FUNCTION_BLOCK FB 52
TITLE = Motor with 6 digital input
//  
//COPYRIGHT:    (C) 1997  BUHLER AG, CH-9240 UZWIL,  SWITZERLAND
//
//PRODUCT:      GCS7
//
//TITLE:        FB 50 MACHINE-CONTROL:Motor with 6 Digital input 
//              GCPROVB Revision >=12
// 
//-------------------------------------------------------------------------
//
//IDENT:        AUTHOR:             DEPT:                       DATE:
//FB50.8.6      A.Egli              BASE                        10-Apr-2008
//              - Init if download DB
//              - Condition MonX.InLocal 
//FB50.8.5      Ph. Engler          GP92                        23-Aug-2007
//              Machine status: StStarting how long the monitoring elements
//FB50.8.5      Ph. Engler          GP92                        23-Aug-2007
//              Machine status: StStarting how long the monitoring elements
//                              aren't in the correct status
//FB50.8.4      A.Egli              CT3                         20-Feb-2006
//              EBM-Test procedure: - Include als the EBMInput to the test
//                                  - Manual and local mode also integrated 
//              (Tested Ph.Engler, GP92,24-Aug-2005 )
//FB50.8.3      A.Egli              CT3                         09-Mar-2005
//              Send CmdFaultReset only with positve edge to elements  
//FB50.8.2      A.Egli              CT3                         20-Sep-2004 
//              Delay time before and between 2 single tests of EBM  
//FB50.8.1      A.Egli              CT3                         20-Jul-2004
//              tmpLenDyn is 12 and not 10
//FB50.8.0      A.Egli              CT3                         25-Mai-2004
//              ParMon4IsSM
//FB50.7.6      A.Egli              CT3                         15-Apr-2004
//              Test with Hardware 
//FB50.7.5      A.Egli              CT3                         18-Mar-2004
//              InpControlEBM 
//FB50.7.4      K. Tischer          CT3                         13-Feb-2004
//              interlocking without Mon1 
//FB50.7.3      K. Tischer          CT3                         30-Jan-2004
//              Correct monitoring Mon4 
//FB50.7.2      K. Tischer          CT3                         14-Jan-2004
//              Revision=11 
//FB50.7.1      K. Tischer          CT3                         02-Dec-2003
//              new 6 DI and supported EBM3003 
//FB50.7.0      K. Tischer          CT3                         01-Dec-2003
//              new 6 DI and supported EBM3003 
//FB50.6.2      A. Egli             CT3                         22-Sep-2003
//              Interlocking Mon4.StFalse when Mon4 is HL
//FB50.6.1      A. Egli             CT3                         16-Mai-2003
//              Interlocking if Mon1 is HL
//              Send CmdOff to Motor
//FB50.6.0      A. Egli             CT3                         17-Jun-2002
//              New Release with one block 
//              Interlocking if Mon1 is HL
//FB50.5.0      A. Egli             CT3                          1-Feb-2002
//              -HLInlet renamed as Mon4
//              -ParMon4StopByFault,ParMon4IsLS
//FB50.4.0      A. Egli             CT3                         15-Jan-2002
//              HLIntet as Warning Element
//FB50.3.1      A. Egli             CT3                         23-Oct-2001
//              Manual Mode: no interlocking with InSeqStop
//FB50.3.0      A. Egli             CT3                         11-Oct-1999
//              Local data reduced 
//FB50.2C       A. Egli             CT3                         03-Juni-1999
//              Manual Mode
//FB50.2B       K. Tischer          MU664                       06-Mrz-1999
//              CC FC2 not UC FC2
//FB50.2A       A. Egli             CT3                         04-Mai-1998
//              StFault = StCode 32
//FB50.1A       A.Egli              AEE61                       5-Jul-1997
//              1st Release in S7
//
//-------------------------------------------------------------------------
//
//PURPOSE:      MANUAL : see [LL.M4IxxMAN]
//
//RESTRICTIONS: S7
//
//              GCPROVB Revision >=5
//-------------------------------------------------------------------------
//
AUTHOR : EA
FAMILY : GCS7LL
NAME : M_6DI
VERSION : 8.6
VAR
  Ma : UDT 20500;
  Mon1 : FB 14;	//Element Mon 1 optional
  Mon2 : FB 14;	//Element Mon 2
  Mon3 : FB 14;	//Element Mon 3 optional
  Mon4 : FB 14;	//Element Mon 4 optional
  Mon5 : FB 14;	//Element Mon 5 optional [7.0]
  Mon6 : FB 14;	//Element Mon 6 optional [7.0]
  Motor : FB 12;	//Element Motor
END_VAR
VAR_TEMP
  tmpFaultStop : BOOL ;
  tmpFaultSum : BOOL ;
  tmpEnable : BOOL ;
  tmpLocal : BOOL ;
  tmpLenDyn : INT ;
  tmpOK : BOOL ;
  tmpTestTime : INT ;
  tmpMonElOk : BOOL ;
END_VAR
BEGIN
NETWORK
TITLE =
      L     12;
      T     #tmpLenDyn;	//[8.1]
NETWORK
TITLE = PC Control
//=== Test Object number =====================
      L     DB3.DBW 50;	//PCControl.ObjectNo
      L     DIW [AR2,P#8.0];	//Input ObjectNo
      <>I;
      JC    aEnd;
//=== Test OType      ========================
      L     2050;	//Input object type
      L     DB3.DBW 48;	//PCControl.ObjectType
      <>I;
      JC    aEnd;
//=== Test Handshake =========================
      A     DB3.DBX 43.3;	// Handshake.FExamine
      JC    aExa;
      A     DB3.DBX 43.0;	// Handshake.FDefineCmd
      O     DB3.DBX 43.1;	// Handshake.FDefinePara
      JC    aCmd;
aIni: L     2;	// FcInit
      UC    FC 3;
      JU    aEnd;
// Write new commands from PC to Interface of group 
aCmd: A     DB3.DBX 53.0;	//Cmd1[8]=CmdOff
      S     DIX [AR2,P#3.0];
      A     DB3.DBX 53.1;	//Cmd1[9]=CmdOn
      S     DIX [AR2,P#3.1];
      A     DB3.DBX 53.2;	//Cmd1[10]=CmdNext
      S     DIX [AR2,P#3.2];
      A     DB3.DBX 53.3;	//Cmd1[11]=CmdFaultReset
      S     DIX [AR2,P#3.3];
      A     DB3.DBX 53.5;	//Cmd1[13]=CmdManualOn
      S     DIX [AR2,P#3.5];
      A     DB3.DBX 52.6;	//Cmd1[6]=CmdManSlowOn
      S     DIX [AR2,P#221.6];
      A     DB3.DBX 52.7;	//Cmd1[7]=CmdManRevOn
      S     DIX [AR2,P#221.7];
      A     DB3.DBX 55.5;	//Cmd2[13]=CmdManualOff
      R     DIX [AR2,P#3.5];
      A     DB3.DBX 54.6;	//Cmd2[6]=CmdManSlowOff
      R     DIX [AR2,P#221.6];
      A     DB3.DBX 54.7;	//Cmd2[7]=CmdManRevOff
      R     DIX [AR2,P#221.7];
      JU    aIni;
aExa: TAR2;	// Address Dynamic datas
      T     DB3.DBD 24;	// -->PCControl.GC.InDynAddr
      L     #tmpLenDyn;	// Length Dynamic data
      T     DB3.DBW 22;	// -->PCControl.GC.InDynLen
      L     0;
      T     DB3.DBD 30;	// -->PCControl.GC.InParaAddr
      T     DB3.DBW 28;	// -->PCControl.GC.InParaLen
      L     1;	// Code FcExamine
      UC    FC 3;
      L     12;	//Revision
      T     DB3.DBW 34;
aEnd: NOP   0;
NETWORK
TITLE = function test [7.0]
      L     720;	//[8.2] 
      T     #tmpTestTime;	//[8.2] 
      AN    DIX [AR2,P#11.5];
      JC    FCT0;
      A     DIX [AR2,P#3.4];
      AN    DIX [AR2,P#3.5];
      =     #tmpLocal;
      L     0;
      L     DIW [AR2,P#6.0];
      >=I;
      O     DIX [AR2,P#3.6];
      R     DIX [AR2,P#4.1];
      R     DIX [AR2,P#4.2];
      R     DIX [AR2,P#4.3];
      R     DIX [AR2,P#3.6];
      L     #tmpTestTime;	//s = 12min 
      JC    FCT;
      AN    DIX [AR2,P#221.2];	//[8.2] 
      AN    DIX [AR2,P#221.5];	//[8.2] 
      AN    DIX [AR2,P#4.3];	//[8.2] 
      L     #tmpTestTime;	//[8.2] 
      JC    FCT;	//[8.2] 
      L     DIW [AR2,P#6.0];
      AN    M 10.5;	// Gr.OutTick1s
      JC    FCT;
      +     -1;
FCT:  T     DIW [AR2,P#6.0];
// function test SM
      L     #tmpTestTime;	//[8.2] 
      L     DIW [AR2,P#6.0];	//[8.2] 
      -I;	//[8.2] 
      L     35;	//[8.2] 
      >=I;	//[8.2] 
      A     DIX [AR2,P#2.6];	//[7.5]
      AN    DIX [AR2,P#4.7];	//[7.5]
      AN    DIX [AR2,P#5.4];	//[7.5]
      O     DIX [AR2,P#4.6];	//[7.5]
      AN    DIX [AR2,P#4.3];
      AN    DIX [AR2,P#15.4];
      AN    DIX [AR2,P#5.0];	//[8.2]
      =     DIX [AR2,P#4.6];
// function test ok SM
      A     DIX [AR2,P#4.6];
      A(;
      ON    DIX [AR2,P#184.6];
      ON    DIX [AR2,P#10.4];
      );
      AN    DIX [AR2,P#2.6];	//[7.5]
      =     #tmpOK;	//[7.5]
      A     #tmpOK;	//[7.5]
      AN    DIX [AR2,P#4.3];	//[7.5]
      S     DIX [AR2,P#4.3];
      S     DIX [AR2,P#2.5];	//[7.5]
      JCN   BTJ1;	//[8.2] 
      L     #tmpTestTime;	//[8.2] s = 12min 
      T     DIW [AR2,P#6.0];	//[8.2] 
BTJ1: NOP   0;	//[8.2] 
// function test BM top
      L     #tmpTestTime;	//[8.2] s = 12min 
      L     DIW [AR2,P#6.0];	//[8.2] 
      -I;	//[8.2] 
      L     5;	//[8.2] 
      >=I;	//[8.2] 
      AN    DIX [AR2,P#4.7];	//[7.5]
      A     DIX [AR2,P#2.6];	//[7.5]
      AN    DIX [AR2,P#5.4];	//[7.5]
      O     DIX [AR2,P#4.4];	//[7.5]
      AN    DIX [AR2,P#4.1];
      A     DIX [AR2,P#4.3];	//[7.6]
      AN    DIX [AR2,P#15.4];
      =     DIX [AR2,P#4.4];
// function test ok
      A     DIX [AR2,P#4.4];
      AN    DIX [AR2,P#48.6];
      AN    DIX [AR2,P#2.6];	//[7.5]
      =     #tmpOK;	//[7.5]
      A     #tmpOK;	//[7.5]
      AN    DIX [AR2,P#4.1];	//[7.5]
      S     DIX [AR2,P#4.1];
      S     DIX [AR2,P#2.5];	//[7.5]
      JCN   BTJ2;	//[8.2] 
      L     #tmpTestTime;	//[8.2] s = 12min 
      T     DIW [AR2,P#6.0];	//[8.2] 
BTJ2: NOP   0;	//[8.2] 
// function test BM Bottom
      L     #tmpTestTime;	//[8.2] s = 12min 
      L     DIW [AR2,P#6.0];	//[8.2] 
      -I;	//[8.2] 
      L     5;	//[8.2] 
      >=I;	//[8.2] 
      A     DIX [AR2,P#2.6];	//[7.5]
      AN    DIX [AR2,P#4.7];	//[7.5]
      AN    DIX [AR2,P#5.4];	//[7.5]
      O     DIX [AR2,P#4.5];	//[7.5]
      AN    DIX [AR2,P#4.2];
      A     DIX [AR2,P#4.1];
      A     DIX [AR2,P#4.3];	//[7.6]
      AN    DIX [AR2,P#15.4];
      =     DIX [AR2,P#4.5];
// function test ok BM Bottom 
      A     DIX [AR2,P#4.5];
      A(;
      ON    DIX [AR2,P#116.6];
      ON    DIX [AR2,P#10.2];
      );
      AN    DIX [AR2,P#2.6];	//[7.5]
      =     #tmpOK;	//[7.5]
      A     #tmpOK;	//[7.5]
      AN    DIX [AR2,P#4.2];	//[7.5]
      S     DIX [AR2,P#4.2];
      S     DIX [AR2,P#2.5];	//[7.5]
FCT0: NOP   0;
NETWORK
TITLE = Interlocking
//===Global Group Orders===
      A     M 12.5;	//Gr.OutManualOn
      S     DIX [AR2,P#3.5];
      A     M 12.4;	//Gr.OutManualOff
      R     DIX [AR2,P#3.5];
      A     DIX [AR2,P#3.5];
      S     M 13.5;	//Gr.InManual
// 
      A     M 12.3;	// OutFaultReset
      S     DIX [AR2,P#3.3];
//--- Fault----
      A     DIX [AR2,P#10.7];
      A     DIX [AR2,P#17.4];
      O     DIX [AR2,P#51.4];
      O     DIX [AR2,P#85.4];
      O(;	//[5.0]
      A     DIX [AR2,P#11.3];	//[5.0]
      O     DIX [AR2,P#11.6];	//[8.0]
      O     DIX [AR2,P#11.5];	//[7.6]
      A     DIX [AR2,P#119.4];	//[5.0]
      );	//[5.0]
      O     DIX [AR2,P#153.4];	//[7.0]
      O     DIX [AR2,P#187.4];	//[7.0]
      =     #tmpFaultStop;
      A     DIX [AR2,P#119.4];	//[4.0]
      AN    DIX [AR2,P#11.2];	//[4.0]
      O     DIX [AR2,P#17.4];
      O     DIX [AR2,P#221.4];
      O     #tmpFaultStop;
      =     #tmpFaultSum;
      A     DIX [AR2,P#119.4];	//[4.0]
      A     DIX [AR2,P#11.2];	//[4.0]
      =     DIX [AR2,P#4.0];	//[4.0]
//--- Motor----
      A     #tmpFaultStop;	//[8.4]
      A     DIX [AR2,P#11.5];	//[8.4]
      A     DIX [AR2,P#219.5];	//[8.4]
      O     DIX [AR2,P#3.0];
      S     DIX [AR2,P#219.0];
//  
      A     DIX [AR2,P#17.2];
      O     DIX [AR2,P#17.3];
      ON    DIX [AR2,P#10.6];	//[6.1]
      ON    DIX [AR2,P#10.7];
      A(;	//[6.0]
      O     DIX [AR2,P#17.0];	//[6.0]
      O     DIX [AR2,P#17.1];	//[6.0]
      ON    DIX [AR2,P#10.5];	//[6.0]
      O     DIX [AR2,P#2.2];	//[6.0]
      );
      ON    DIX [AR2,P#10.0];	//[7.4]
      A(;
      A     DIX [AR2,P#11.5];	//[7.6]
      O     DIX [AR2,P#51.2];
      O     DIX [AR2,P#51.3];
      ON    DIX [AR2,P#11.0];
      );
      A(;
      A     DIX [AR2,P#11.5];	//[7.6]
      O     DIX [AR2,P#85.2];
      O     DIX [AR2,P#85.3];
      ON    DIX [AR2,P#10.1];
      ON    DIX [AR2,P#11.1];
      );
      A(;
      A     DIX [AR2,P#11.5];	//[7.6]
      O     DIX [AR2,P#119.2];	//[6.2]
      O     DIX [AR2,P#119.3];	//[6.2]
      A     DIX [AR2,P#11.4];	//[6.2]
      O(;	//[6.2]
      A     DIX [AR2,P#119.0];	//[6.2]
      O     DIX [AR2,P#119.1];	//[6.2]
      O     DIX [AR2,P#2.2];	//[6.2]
      AN    DIX [AR2,P#11.4];	//[6.2]
      );	//[6.2]
      ON    DIX [AR2,P#11.3];	//[6.2]
      O     DIX [AR2,P#11.6];	//[8.0]
      ON    DIX [AR2,P#10.2];	//[6.2]
      );	//[6.2]
      A(;	//[7.0]
      A     DIX [AR2,P#11.5];	//[7.6]
      O     DIX [AR2,P#153.2];	//[7.0]
      O     DIX [AR2,P#153.3];	//[7.0]
      ON    DIX [AR2,P#10.3];	//[7.0]
      );	//[7.0]
      A(;	//[7.0]
      A     DIX [AR2,P#11.5];	//[7.6]
      O     DIX [AR2,P#187.2];	//[7.0]
      O     DIX [AR2,P#187.3];	//[7.0]
      ON    DIX [AR2,P#10.4];	//[7.0]
      );	//[7.0]
      =     #tmpEnable;	//[4.0]
//Set speed if manual mode without interlocking                   
      AN    DIX [AR2,P#230.1];
      ON    DIX [AR2,P#3.5];
      O     DIX [AR2,P#219.5];
      JC    inJo;
      A     DIX [AR2,P#221.6];
      =     DIX [AR2,P#218.2];
inJo: A(;
      AN    DIX [AR2,P#230.1];
      AN    DIX [AR2,P#221.7];
      ON    DIX [AR2,P#3.5];
      A     DIX [AR2,P#2.1];
      O;
      A     DIX [AR2,P#3.5];
      A     DIX [AR2,P#230.1];
      AN    DIX [AR2,P#221.7];
      );
      AN    DIX [AR2,P#2.7];
      AN    #tmpFaultStop;
      AN    DIX [AR2,P#3.0];
      A     #tmpEnable;	//[4.0]
      =     DIX [AR2,P#218.1];
      A(;
      AN    DIX [AR2,P#230.1];
      A     DIX [AR2,P#221.7];
      ON    DIX [AR2,P#3.5];
      A     DIX [AR2,P#2.0];
      O;
      A     DIX [AR2,P#3.5];
      A     DIX [AR2,P#230.1];
      A     DIX [AR2,P#221.7];
      );
      AN    DIX [AR2,P#2.7];
      AN    #tmpFaultStop;
      AN    DIX [AR2,P#3.0];
      A     #tmpEnable;	//[4.0]
      =     DIX [AR2,P#218.0];
      A     DIX [AR2,P#3.2];
      AN    DIX [AR2,P#3.5];
      O;
      A     DIX [AR2,P#3.5];
      A     DIX [AR2,P#3.1];
      S     DIX [AR2,P#219.2];
      A     DIX [AR2,P#3.7];
      AN    DIX [AR2,P#3.5];	// [3.1]
      =     DIX [AR2,P#219.7];
//--- Local mode --
      A     DIX [AR2,P#3.4];
      AN    DIX [AR2,P#3.5];
      =     #tmpLocal;
      A     #tmpLocal;
      =     DIX [AR2,P#219.4];
      AN    #tmpFaultStop;	//[8.6]
      O     #tmpLocal;	//[8.6]
      AN    DIX [AR2,P#218.6];	//[8.4]
      AN    DIX [AR2,P#218.5];	//[8.4]
      AN    DIX [AR2,P#219.5];	//[8.4]
      A(;	//[8.6]
      L     DIW [AR2,P#216.0];	//[8.6]
      L     0;	//[8.6]
      ==I;	//[8.6]
      O     DIX [AR2,P#221.0];	//[7.6]
      );	//[8.6]
      ON    DIX [AR2,P#11.5];	//[7.6]
      A     #tmpLocal;	//[7.6]
      =     DIX [AR2,P#117.4];	//[7.6]
      AN    #tmpFaultStop;	//[8.6]
      O     #tmpLocal;	//[8.6]
      AN    DIX [AR2,P#218.6];	//[8.4]
      AN    DIX [AR2,P#218.5];	//[8.4]
      AN    DIX [AR2,P#219.5];	//[8.4]
      ON    DIX [AR2,P#11.5];	//[8.4]
      A     #tmpLocal;
      A(;	//[8.6]
      L     DIW [AR2,P#216.0];	//[8.6]
      L     0;	//[8.6]
      ==I;	//[8.6]
      O     DIX [AR2,P#221.0];	//[7.6]
      );	//[8.6]
      =     DIX [AR2,P#15.4];
      =     DIX [AR2,P#49.4];
      =     DIX [AR2,P#83.4];
      =     DIX [AR2,P#151.4];	//[7.0]
      =     DIX [AR2,P#185.4];	//[7.0]
//--- Monitoring
      A     DIX [AR2,P#10.6];
      O     DIX [AR2,P#221.2];
      O     DIX [AR2,P#221.5];
      AN    DIX [AR2,P#10.5];
      =     DIX [AR2,P#14.0];
      A     DIX [AR2,P#10.5];
      AN    DIX [AR2,P#2.2];
      =     DIX [AR2,P#14.1];
//Mon2
      A     DIX [AR2,P#4.4];	//[7.0]
      =     DIX [AR2,P#48.1];	//[7.0]
      A     DIX [AR2,P#11.0];
      O     DIX [AR2,P#221.2];
      O     DIX [AR2,P#221.5];
      O     DIX [AR2,P#11.5];	//[7.3]
      AN    DIX [AR2,P#4.5];	//[7.0]
      AN    DIX [AR2,P#48.1];	//[7.0]
      =     DIX [AR2,P#48.0];
//Mon3
      A     DIX [AR2,P#4.4];	//[7.0]
      A     DIX [AR2,P#10.1];	//[7.0]
      =     DIX [AR2,P#82.1];	//[7.0]
      A     DIX [AR2,P#11.1];
      O     DIX [AR2,P#221.2];
      O     DIX [AR2,P#221.5];
      O     DIX [AR2,P#11.5];	//[7.3]
      AN    DIX [AR2,P#4.5];	//[7.0]
      AN    DIX [AR2,P#82.1];	//[7.0]
      =     DIX [AR2,P#82.0];
//Mon4
      A     DIX [AR2,P#11.2];	//[4.0]
      O     DIX [AR2,P#11.4];	//[5.0]
      O     DIX [AR2,P#11.5];	//[7.3]
      O(;	//[7.3]
      O     DIX [AR2,P#221.2];	//[7.0]
      O     DIX [AR2,P#221.5];	//[7.0]
      A     DIX [AR2,P#11.6];	//[8.0]
      );	//[7.3]
      AN    DIX [AR2,P#4.4];	//[7.0]
      AN    DIX [AR2,P#4.5];	//[7.0]
      A     DIX [AR2,P#10.2];	//[7.0]
      =     DIX [AR2,P#116.0];	//[4.0]
      A(;	//[8.0]
      AN    DIX [AR2,P#116.0];	//[7.0]
      AN    DIX [AR2,P#11.5];	//[7.0]
      A     DIX [AR2,P#10.2];	//[7.0]
      O;
      A     DIX [AR2,P#4.5];	//[7.0]
      A     DIX [AR2,P#10.2];	//[7.0]
      );	//[8.0]
      AN    DIX [AR2,P#11.6];	//[8.0]
      =     DIX [AR2,P#116.1];
//Mon5
      A     DIX [AR2,P#4.5];	//[7.0]
      A     DIX [AR2,P#10.3];	//[7.0]
      =     DIX [AR2,P#150.1];	//[7.0]
      A     DIX [AR2,P#221.2];	//[7.0]
      O     DIX [AR2,P#221.5];	//[7.0]
      O     DIX [AR2,P#11.5];	//[7.3]
      AN    DIX [AR2,P#4.4];	//[7.0]
      AN    DIX [AR2,P#150.1];	//[7.0]
      =     DIX [AR2,P#150.0];	//[7.0]
//Mon6
      A     DIX [AR2,P#4.6];	//[7.0]
      A     DIX [AR2,P#10.4];	//[7.0]
      =     DIX [AR2,P#184.1];	//[7.0]
      A     DIX [AR2,P#221.2];	//[7.0]
      O     DIX [AR2,P#221.5];	//[7.0]
      O     DIX [AR2,P#11.5];	//[7.3]
      AN    DIX [AR2,P#184.1];	//[7.0]
      =     DIX [AR2,P#184.0];	//[7.0]
//--- Fault Reset -------------
      A     DIX [AR2,P#3.3];
      FP    DIX [AR2,P#2.4];	//[8.3]
      S     DIX [AR2,P#117.3];
      S     DIX [AR2,P#219.3];
      S     DIX [AR2,P#15.3];
      S     DIX [AR2,P#49.3];
      S     DIX [AR2,P#83.3];
      S     DIX [AR2,P#151.3];	//[7.0]
      S     DIX [AR2,P#185.3];	//[7.0]
NETWORK
TITLE = Call Digital Input: Monitor B1
      AN    DIX [AR2,P#10.0];	//[7.0]
      JC    Mon2;	//[7.0]
      BLD   14;
      =     L 15.0;
      L     DINO;
      T     LW 13;
      CDB;
      OPN   DI [LW 13];
      TAR2  LD 9;
      +AR2  P#12.0;
      UC    FB 14;
      LAR2  LD 9;
      CDB;
      BLD   15;
NETWORK
TITLE = Call Digital Input: Monitor B2
Mon2: A     DIX [AR2,P#2.6];	//[8.4]
      A     DIX [AR2,P#4.4];	//[8.4]
      A     DIX [AR2,P#11.5];	//[8.4]
      O     DIX [AR2,P#48.6];	//[8.4]
      =     DIX [AR2,P#48.6];	//[8.4]
      BLD   14;
      =     L 15.0;
      L     DINO;
      T     LW 13;
      CDB;
      OPN   DI [LW 13];
      TAR2  LD 9;
      +AR2  P#46.0;
      UC    FB 14;
      LAR2  LD 9;
      CDB;
      BLD   15;
NETWORK
TITLE = Call Digital Input: Monitor B3
      AN    DIX [AR2,P#10.1];
      JC    Mon4;	//[7.0]
      A     DIX [AR2,P#2.6];	//[8.4]
      A     DIX [AR2,P#4.4];	//[8.4]
      A     DIX [AR2,P#11.5];	//[8.4]
      O     DIX [AR2,P#82.6];	//[8.4]
      =     DIX [AR2,P#82.6];	//[8.4]
      BLD   14;
      =     L 15.0;
      L     DINO;
      T     LW 13;
      CDB;
      OPN   DI [LW 13];
      TAR2  LD 9;
      +AR2  P#80.0;
      UC    FB 14;
      LAR2  LD 9;
      CDB;
      BLD   15;
NETWORK
TITLE = Call Digital Input: Mon4
Mon4: AN    DIX [AR2,P#10.2];	//[7.0]
      JC    Mon5;
      A     DIX [AR2,P#2.6];	//[8.4]
      A     DIX [AR2,P#4.5];	//[8.4]
      A     DIX [AR2,P#11.5];	//[8.4]
      O     DIX [AR2,P#116.6];	//[8.4]
      =     DIX [AR2,P#116.6];	//[8.4]
      BLD   14;
      =     L 15.0;
      L     DINO;
      T     LW 13;
      CDB;
      OPN   DI [LW 13];
      TAR2  LD 9;
      +AR2  P#114.0;
      UC    FB 14;
      LAR2  LD 9;
      CDB;
      BLD   15;
NETWORK
TITLE = Call Digital Input: Mon5  [7.0]
Mon5: AN    DIX [AR2,P#10.3];	//[7.0]
      JC    Mon6;	//[7.0]
      A     DIX [AR2,P#2.6];	//[8.4]
      A     DIX [AR2,P#4.5];	//[8.4]
      A     DIX [AR2,P#11.5];	//[8.4]
      O     DIX [AR2,P#150.6];	//[8.4]
      =     DIX [AR2,P#150.6];	//[8.4]
      BLD   14;	//[7.0]
      =     L 15.0;
      L     DINO;
      T     LW 13;
      CDB;
      OPN   DI [LW 13];
      TAR2  LD 9;
      +AR2  P#148.0;
      UC    FB 14;
      LAR2  LD 9;
      CDB;
      BLD   15;
NETWORK
TITLE = Call Digital Input: Mon6 [7.0]
Mon6: AN    DIX [AR2,P#10.4];	//[7.0]
      JC    Mo;	//[7.0]
      A     DIX [AR2,P#2.6];	//[8.4]
      A     DIX [AR2,P#4.6];	//[8.4]
      A     DIX [AR2,P#11.5];	//[8.4]
      O     DIX [AR2,P#184.6];	//[8.4]
      =     DIX [AR2,P#184.6];	//[8.4]
      BLD   14;	//[7.0]
      =     L 15.0;
      L     DINO;
      T     LW 13;
      CDB;
      OPN   DI [LW 13];
      TAR2  LD 9;
      +AR2  P#182.0;
      UC    FB 14;
      LAR2  LD 9;
      CDB;
      BLD   15;
NETWORK
TITLE = Call Motor
Mo:   BLD   14;
      =     L 15.0;
      L     DINO;
      T     LW 13;
      CDB;
      OPN   DI [LW 13];
      TAR2  LD 9;
      +AR2  P#216.0;
      UC    FB 12;
      LAR2  LD 9;
      CDB;
      BLD   15;
NETWORK
TITLE = State
// Stopped
      A(;	//[8.5]
      A     DIX [AR2,P#17.2];	//[8.5]
      AN    DIX [AR2,P#10.5];	//[8.5]
      O;	//[8.5]
      A     DIX [AR2,P#17.0];	//[8.5]
      A     DIX [AR2,P#10.5];	//[8.5]
      ON    DIX [AR2,P#10.7];	//[8.5]
      ON    DIX [AR2,P#10.0];	//[8.5]
      );	//[8.5]
      A     DIX [AR2,P#51.2];	//[8.5]
      A(;	//[8.5]
      A     DIX [AR2,P#85.2];	//[8.5]
      ON    DIX [AR2,P#10.1];	//[8.5]
      );	//[8.5]
      A(;	//[8.5]
      A     DIX [AR2,P#11.4];	//[8.5]
      O     DIX [AR2,P#11.6];	//[8.5]
      A     DIX [AR2,P#119.2];	//[8.5]
      O;	//[8.5]
      A     DIX [AR2,P#119.0];	//[8.5]
      AN    DIX [AR2,P#11.4];	//[8.5]
      AN    DIX [AR2,P#11.6];	//[8.5]
      AN    DIX [AR2,P#11.5];	//[8.5]
      O     DIX [AR2,P#11.2];	//[8.5]
      ON    DIX [AR2,P#11.3];	//[8.5]
      ON    DIX [AR2,P#10.2];	//[8.5]
      );	//[8.5]
      A(;	//[8.5]
      A     DIX [AR2,P#153.2];	//[8.5]
      ON    DIX [AR2,P#10.3];	//[8.5]
      );	//[8.5]
      A(;	//[8.5]
      A     DIX [AR2,P#187.2];	//[8.5]
      ON    DIX [AR2,P#10.4];	//[8.5]
      );	//[8.5]
      =     #tmpMonElOk;	//[8.5]
// Stopped
      A     DIX [AR2,P#221.0];
      AN    #tmpFaultSum;
      AN    DIX [AR2,P#2.7];
      =     DIX [AR2,P#5.0];
// Locked 
      A     DIX [AR2,P#221.0];
      AN    #tmpFaultSum;
      A     DIX [AR2,P#2.7];
      =     DIX [AR2,P#5.6];
// Starting
      O     DIX [AR2,P#221.2];	//[8.5]
      O     DIX [AR2,P#221.5];	//[8.5]
      AN    #tmpMonElOk;	//[8.5]
      AN    DIX [AR2,P#5.2];	//[8.5]
      AN    DIX [AR2,P#5.5];	//[8.5]
      O     DIX [AR2,P#221.1];
      AN    #tmpFaultSum;
      =     DIX [AR2,P#5.1];
// StartedFwd
      A     DIX [AR2,P#221.2];
      AN    DIX [AR2,P#5.1];	//[8.5]
      AN    #tmpFaultSum;
      =     DIX [AR2,P#5.2];
// StartedRev
      A     DIX [AR2,P#221.5];
      AN    DIX [AR2,P#5.1];	//[8.5]
      AN    #tmpFaultSum;
      =     DIX [AR2,P#5.5];
// Stopping
      A     DIX [AR2,P#221.3];
      AN    #tmpFaultSum;
      =     DIX [AR2,P#5.3];
// Fault
      A     #tmpFaultSum;
      =     DIX [AR2,P#5.4];
NETWORK
TITLE = Global End
      NOP   0;
//--------------------------------
//Pulse length OutpFaultReset is 500ms
      A     M 10.5;	//[7.0]
      R     DIX [AR2,P#4.7];	//[7.0]
//--------------------------------
//Set OutpFaultReset
// - with tick  "GCS7_Gr_OutTick1s"
// - Negativ flag of Ma.InpControlEBM during test
      AN    DIX [AR2,P#2.6];	//[7.6]
      A     DIX [AR2,P#11.5];	//[7.6]
      O     DIX [AR2,P#5.4];	//[7.0]
      A     M 10.5;	//[7.0]
      A     DIX [AR2,P#3.3];	//[7.0]
      O;
      A     DIX [AR2,P#2.5];	//[7.5]
      AN    DIX [AR2,P#5.4];	//[7.5]
      S     DIX [AR2,P#4.7];	//[7.0]
      R     DIX [AR2,P#3.3];	//[7.5]
      A     DIX [AR2,P#4.7];	//[7.5]
      A     DIX [AR2,P#2.6];	//[7.6]
      R     DIX [AR2,P#2.5];	//[7.5]
//--------------------------------
//Reset OutpFaultReset immediatly when InpControlEBM is ok
      A     DIX [AR2,P#2.6];	//[7.6]
      O     DIX [AR2,P#5.4];	//[7.6]
      A     DIX [AR2,P#2.5];	//[7.5]
      R     DIX [AR2,P#2.5];	//[7.5]
      R     DIX [AR2,P#4.7];	//[7.0]
//--------------------------------
//Reset  CmdFaultReset when no fault
      A     DIX [AR2,P#2.6];	//[7.6]
      ON    DIX [AR2,P#11.5];	//[7.6]
      AN    DIX [AR2,P#5.4];	//[7.0]
      R     DIX [AR2,P#3.3];	//[7.5]
//--------------------------------
//Init commands
      CLR;	//---Clear all commands
      =     DIX [AR2,P#3.1];
      =     DIX [AR2,P#3.0];
      =     DIX [AR2,P#3.2];
NETWORK
TITLE = State Code
// Same as motor
      A     DIX [AR2,P#5.6];
      L     8;	//  StCode=Locked
      JC    Code;
      L     DIW [AR2,P#216.0];	// StCode=Motor
      AN    DIX [AR2,P#5.4];
      JC    Code;
      L     32;	// StCode=Fault
Code: L     DIW [AR2,P#0.0];	// Old state code
      TAK;
      T     DIW [AR2,P#0.0];	// Save state code
      <>I;
      L     3;
      CC    FC 2;	//Set change bit
END_FUNCTION_BLOCK

FUNCTION_BLOCK "G270M_Code"	// FB 370
TITLE = G270M AIR SHUT SLIDE KILN 1
//COPYRIGHT:    (C) 2009  BUHLER AG, CH-9240 UZWIL, SWITZERLAND
//
//PRODUCT:      WinCoS_BIW01_09
//
//TITLE:        AIR SHUT SLIDE KILN 1
//                Machine group control
//                Maschinengruppensteuerung
// 
//--------------------------------------------------------------------------------
// 
//IDENT:        AUTHOR:             DEPT:                              DATE:
// 
//P01_FB370.1.0 K.Renz              CSB41                              06.Okt.2009
//             1st Release
// 
//--------------------------------------------------------------------------------
// 
//PURPOSE: 
// 
//MANUAL : 
// 
//RESTRICTIONS: 
// 
//--------------------------------------------------------------------------------
//
AUTHOR : KR
FAMILY : USW
VERSION : 9.9
VAR
  Gr : FB 10;	//Standard interface to group
  InOutValue1 : DINT ;	//Data for user
  InOutValue2 : DINT ;	//Data for user
  OutWayConflict : BOOL ;	//Data for user
  OutSelectionOk : BOOL ;	//Data for user
  CmdNewValue : BOOL ;	//Data for user
  CmdNewJob : BOOL ;	//Data for user
  OutCodeOK : BOOL ;	//Data for user
  InEndOfJob : BOOL ;	//Data for user
  staWayOk : BOOL ;	//Data for user
  EdgeStartRelease : BOOL ;	//Data for user
  USW8 : BOOL ;	//Data for user
  USW9 : BOOL ;	//Data for user
  USW10 : BOOL ;	//Data for user
  USW11 : BOOL ;	//Data for user
  USW12 : BOOL ;	//Data for user
  USW13 : BOOL ;	//Data for user
  USW14 : BOOL ;	//Data for user
  USW15 : BOOL ;	//Data for user
  A_3101_MXZ01 : FB 13;	// VLS
END_VAR
VAR_TEMP
  tmpEnable : BOOL ;
  tmpFlag : BOOL ;
  tmpCmdNext : BOOL ;
  tmpLocal : BOOL ;
  tmpAspOk : BOOL ;
  tmpHWStop : BOOL ;
  tmpInstanzDBNo : INT ;
END_VAR
BEGIN
NETWORK
TITLE =
NETWORK
TITLE = Read command from group control
//Parameter
      SET;
      S     DB9.DBX 83.5;
      R     DB9.DBX 123.5;
      R     DB9.DBX 163.5;
      R     DB9.DBX 43.5;
      R     DB9.DBX 203.5;
      S     DIX [AR2,P#32.0];
      R     DIX [AR2,P#32.1];
      R     DIX [AR2,P#32.2];
//Command
      A     DB9.DBX 323.5;
      =     DIX [AR2,P#14.0];
      A     DB9.DBX 283.5;
      =     DIX [AR2,P#15.4];
      A     DB9.DBX 403.5;
      R     DB9.DBX 403.5;
      S     DIX [AR2,P#15.3];
      A     DB9.DBX 363.5;
      R     DB9.DBX 363.5;
      S     DIX [AR2,P#15.2];
      A     DB9.DBX 443.5;
      AN    DIX [AR2,P#15.5];
      S     DIX [AR2,P#14.7];
      A     DB9.DBX 443.5;
      R     DB9.DBX 443.5;
//      U     "GCS7_GrCtrlDB".CmdManualOff[270]
//      O     "GCS7_GrCtrlDB".OutOccupied[270]
//      R     "GCS7_GrCtrlDB".CmdManualOff[270]
//      S     #Gr.CmdManualOff
      A     DB9.DBX 763.5;
      R     DB9.DBX 763.5;
      S     DIX [AR2,P#14.1];
//Init Line Number
      A     DB9.DBX 203.5;
      JCN   WE00;
      L     0;
      T     DIW [AR2,P#24.0];
WE00: NOP   0;
NETWORK
TITLE = Call Methode Control
// 1. Handle Interface PCControl      
// 2. Prepare mode --> ModePassive,ModeActive,ModeIdling      
// 3. Reset global flags of the group
      BLD   14;
      =     L 10.0;
      L     DINO;
      T     LW 8;
      CDB;
      OPN   DI [LW 8];
      TAR2  LD 4;
      L     1;
      T     DIW [AR2,P#0.0];
      +AR2  P#0.0;
      UC    FB 10;
      LAR2  LD 4;
      CDB;
      BLD   15;
NETWORK
TITLE = Restart Idling Time
      L     DIW [AR2,P#36.0];
      L     2;
      >=I;
      JC    IdTm;
      T     DIW [AR2,P#36.0];
IdTm: NOP   0;
//      CLR   
      A     DIX [AR2,P#65.5];
      AN    DIX [AR2,P#15.4];
      S     DIX [AR2,P#14.2];
NETWORK
TITLE = Prepare global flags
NETWORK
TITLE = Set Pattern (Target position)
NETWORK
TITLE = Interlocking WayOk
NETWORK
TITLE = Interlocking Autostart
      CLR;
      R     DIX [AR2,P#18.4];
NETWORK
TITLE = Interlocking Enable
      A     DIX [AR2,P#14.0];
      =     DIX [AR2,P#18.0];
NETWORK
TITLE = Interlocking Next
      A     DIX [AR2,P#15.2];
      A     DIX [AR2,P#18.4];
      AN    DIX [AR2,P#19.6];
      =     #tmpCmdNext;
NETWORK
TITLE = Interlocking Local / HWStop
      A     DB50.DBX 32.3;
      =     #tmpHWStop;
      A     DIX [AR2,P#16.0];
      O     #tmpHWStop;
      =     #tmpLocal;
NETWORK
TITLE = =A-3101-MXZ01 : OUTLET FLAP DRIVE 
      NOP   0;
//-InLocal---
      A     #tmpLocal;
      A     DIX [AR2,P#65.0];
      =     DIX [AR2,P#63.4];
//-Interlocking---
      A     DB922.DBX 406.0;	// Step loading
//MW 2010.04.08
      A     DIX [AR2,P#18.0];
      =     DIX [AR2,P#62.1];
      NOT;
      =     DIX [AR2,P#62.0];
      SET;
      S     DIX [AR2,P#63.2];
      A     DIX [AR2,P#19.7];
      A     DIX [AR2,P#65.0];
      =     DIX [AR2,P#63.7];
// 
//-Read inputs---
      A     I 908.0;
      =     DIX [AR2,P#62.5];
      A     I 908.1;
      =     DIX [AR2,P#62.6];
      X     Q 904.0;
      X     I 904.0;
      O;
      X     Q 904.1;
      X     I 904.1;
      =     DIX [AR2,P#62.7];
      A     DB50.DBX 32.3;
      =     DIX [AR2,P#64.0];
      A     DB51.DBX 11.2;
      =     DIX [AR2,P#64.1];
// 
//-Set Parameters---
// 
//-Call object control---
      BLD   14;
// 
//-Write outputs---
      =     L 10.0;
      L     DINO;
      T     LW 8;
      CDB;
      OPN   DI [LW 8];
      TAR2  LD 4;
      +AR2  P#60.0;
      UC    FB 13;
      LAR2  LD 4;
      CDB;
      BLD   15;
      A     DIX [AR2,P#64.5];
      =     Q 904.0;
      A     DIX [AR2,P#64.6];
      =     Q 904.1;
NETWORK
TITLE = Test Fault
      A     DIX [AR2,P#65.4];
      =     DIX [AR2,P#19.2];
NETWORK
TITLE = Test Warning
      CLR;
      =     DIX [AR2,P#17.6];
NETWORK
TITLE = Test Stopped
      A     DIX [AR2,P#65.0];
      AN    DIX [AR2,P#19.2];
      =     DIX [AR2,P#19.0];
NETWORK
TITLE = Test Started
      A     DIX [AR2,P#65.2];
      AN    DIX [AR2,P#19.0];
      AN    DIX [AR2,P#19.2];
      =     DIX [AR2,P#19.1];
NETWORK
TITLE = Enable Previous Group
      A     DIX [AR2,P#19.1];
      =     DIX [AR2,P#18.7];
NETWORK
TITLE = Call Methode State
//1. Make State of the group: This function use the signals:
//        Gr.VarStopped, Gr.VarStarted, Gr.VarFault
//2.Reset Commands to group: e.g.CmdFaultReset
      BLD   14;
      =     L 10.0;
      L     DINO;
      T     LW 8;
      CDB;
      OPN   DI [LW 8];
      TAR2  LD 4;
      L     2;
      T     DIW [AR2,P#0.0];
      +AR2  P#0.0;
      UC    FB 10;
      LAR2  LD 4;
      CDB;
      BLD   15;
NETWORK
TITLE = Init
      SET;
      R     DIX [AR2,P#58.2];
      R     DIX [AR2,P#58.3];
NETWORK
TITLE = Write data to group control
      A     DIX [AR2,P#17.0];
      =     DB9.DBX 483.5;
      A     DIX [AR2,P#17.2];
      =     DB9.DBX 523.5;
      A     DIX [AR2,P#17.4];
      =     DB9.DBX 563.5;
      A     DIX [AR2,P#17.6];
      =     DB9.DBX 603.5;
      A     DIX [AR2,P#18.5];
      =     DB9.DBX 643.5;
      A     DIX [AR2,P#18.2];
      =     DB9.DBX 883.5;
      A     DIX [AR2,P#18.3];
      =     DB9.DBX 843.5;
      A     DIX [AR2,P#17.5];
      =     DB9.DBX 803.5;
      A     DIX [AR2,P#18.4];
      =     DB9.DBX 923.5;
      A     DIX [AR2,P#19.3];
      =     DB9.DBX 963.5;
NETWORK
TITLE = End of block
      BE;
END_FUNCTION_BLOCK

FUNCTION_BLOCK "G271M_Code"	// FB 371
TITLE = G271M FAN KILN 1
//COPYRIGHT:    (C) 2009  BUHLER AG, CH-9240 UZWIL, SWITZERLAND
//
//PRODUCT:      WinCoS_BIW01_09
//
//TITLE:        FAN KILN 1
//                Machine group control
//                Maschinengruppensteuerung
// 
//--------------------------------------------------------------------------------
// 
//IDENT:        AUTHOR:             DEPT:                              DATE:
// 
//P01_FB371.1.0 K.Renz              CSB41                              13.Jan.2010
//             1st Release
// 
//--------------------------------------------------------------------------------
// 
//PURPOSE: 
// 
//MANUAL : 
// 
//RESTRICTIONS: 
// 
//--------------------------------------------------------------------------------
//
AUTHOR : KR
FAMILY : USW
VERSION : 9.9
VAR
  Gr : FB 10;	//Standard interface to group
  InOutValue1 : DINT ;	//Data for user
  InOutValue2 : DINT ;	//Data for user
  OutWayConflict : BOOL ;	//Data for user
  OutSelectionOk : BOOL ;	//Data for user
  CmdNewValue : BOOL ;	//Data for user
  CmdNewJob : BOOL ;	//Data for user
  OutCodeOK : BOOL ;	//Data for user
  InEndOfJob : BOOL ;	//Data for user
  staWayOk : BOOL ;	//Data for user
  EdgeStartRelease : BOOL ;	//Data for user
  USW8 : BOOL ;	//Data for user
  USW9 : BOOL ;	//Data for user
  USW10 : BOOL ;	//Data for user
  USW11 : BOOL ;	//Data for user
  USW12 : BOOL ;	//Data for user
  USW13 : BOOL ;	//Data for user
  USW14 : BOOL ;	//Data for user
  USW15 : BOOL ;	//Data for user
  A_3125_KCU04AI1 : FB 19;	// AnaInp
  A_3125_KCU04AI2 : FB 19;	// AnaInp
  A_3125_BTE05 : FB 19;	// AnaInp
  A_3125_BTE06 : FB 19;	// AnaInp
  A_3125_MXZ01MA : FB 1018;	// Motor+6DI
  A_3125_TSC01_COM : FB 1816;	// FU_Siemens
  A_3125_TSC01_AC : FB 19;	// AnaInp
  A_3125_TSC01_AF : FB 19;	// AnaInp
  A_3125_TSC01_AT : FB 19;	// AnaInp
  A_3125_TSC01_AP : FB 19;	// AnaInp
  A_3126_KCU04AI1 : FB 19;	// AnaInp
  A_3126_KCU04AI2 : FB 19;	// AnaInp
  A_3126_BTE05 : FB 19;	// AnaInp
  A_3126_BTE06 : FB 19;	// AnaInp
  A_3126_MXZ01MA : FB 1019;	// Motor+6DI
  A_3126_TSC01_COM : FB 1816;	// FU_Siemens
  A_3126_TSC01_AC : FB 19;	// AnaInp
  A_3126_TSC01_AF : FB 19;	// AnaInp
  A_3126_TSC01_AP : FB 19;	// AnaInp
  A_3126_TSC01_AT : FB 19;	// AnaInp
  A_3125_TSC01 : FB 14;	// DigInpCont
  A_3126_TSC01 : FB 14;	// DigInpCont
END_VAR
VAR_TEMP
  tmpEnable : BOOL ;
  tmpFlag : BOOL ;
  tmpCmdNext : BOOL ;
  tmpLocal : BOOL ;
  tmpAspOk : BOOL ;
  tmpHWStop : BOOL ;
  tmpInstanzDBNo : INT ;
END_VAR
BEGIN
NETWORK
TITLE =
NETWORK
TITLE = Read command from group control
//Parameter
      SET;
      S     DB9.DBX 83.6;
      R     DB9.DBX 123.6;
      R     DB9.DBX 163.6;
      R     DB9.DBX 43.6;
      R     DB9.DBX 203.6;
      S     DIX [AR2,P#32.0];
      R     DIX [AR2,P#32.1];
      R     DIX [AR2,P#32.2];
//Command
      A     DB9.DBX 323.6;
      =     DIX [AR2,P#14.0];
      A     DB9.DBX 283.6;
      =     DIX [AR2,P#15.4];
      A     DB9.DBX 403.6;
      R     DB9.DBX 403.6;
      S     DIX [AR2,P#15.3];
      A     DB9.DBX 363.6;
      R     DB9.DBX 363.6;
      S     DIX [AR2,P#15.2];
      A     DB9.DBX 443.6;
      AN    DIX [AR2,P#15.5];
      S     DIX [AR2,P#14.7];
      A     DB9.DBX 443.6;
      R     DB9.DBX 443.6;
//      U     "GCS7_GrCtrlDB".CmdManualOff[271]
//      O     "GCS7_GrCtrlDB".OutOccupied[271]
//      R     "GCS7_GrCtrlDB".CmdManualOff[271]
//      S     #Gr.CmdManualOff
      A     DB9.DBX 763.6;
      R     DB9.DBX 763.6;
      S     DIX [AR2,P#14.1];
//Init Line Number
      A     DB9.DBX 203.6;
      JCN   WE00;
      L     0;
      T     DIW [AR2,P#24.0];
WE00: NOP   0;
NETWORK
TITLE = Call Methode Control
// 1. Handle Interface PCControl      
// 2. Prepare mode --> ModePassive,ModeActive,ModeIdling      
// 3. Reset global flags of the group
      BLD   14;
      =     L 10.0;
      L     DINO;
      T     LW 8;
      CDB;
      OPN   DI [LW 8];
      TAR2  LD 4;
      L     1;
      T     DIW [AR2,P#0.0];
      +AR2  P#0.0;
      UC    FB 10;
      LAR2  LD 4;
      CDB;
      BLD   15;
NETWORK
TITLE = Restart Idling Time
      L     DIW [AR2,P#36.0];
      L     2;
      >=I;
      JC    IdTm;
      T     DIW [AR2,P#36.0];
IdTm: NOP   0;
      CLR;
      S     DIX [AR2,P#14.2];
NETWORK
TITLE = Prepare global flags
NETWORK
TITLE = Set Pattern (Target position)
      A     DIX [AR2,P#15.5];
      JC    ILO6;
// Drehzahlabsenkung wenn die andere Horde im Cooling ist
// und die Temperatur unter der eigenen Horde 5°C > als T[Soll] 
//      U     "MAL1S033Par".Par.FlagProcess.Cooling_Activ
//      U     "G276M".USW8                // Temperatur unter der Horde 5°C > T[Soll]
//      L     50                          // 50%
//      SPB   En06
      L     DB922.DBW 228;
//      U     "G275M".USW8                // Drehzahlverrinderung bei offenen Bypassklappen
//      SPBN  En06
//      L     DB799.DBW   26              // Sollwert vom LS
//      -I    
      JU    En06;
ILO6: NOP   0;
      L     DB922.DBW 284;
En06: NOP   0;
      L     100;
      *I;
      T     DIW [AR2,P#666.0];	// xxx.xx%
      T     DIW [AR2,P#1660.0];	// xxx.xx%
NETWORK
TITLE = Interlocking WayOk
NETWORK
TITLE = Interlocking Autostart
      CLR;
      R     DIX [AR2,P#18.4];
NETWORK
TITLE = Interlocking Enable
// (network holds code this reader does not know; not shown)
//--------------------- Ein-Hordenbetrieb ----------------------------//
// Luft-Eintritt
// Luft-Austritt
//---------------------- Zwei-Hordenbetrieb --------------------------//
// Luft-Eintritt
//MW 2010.04.29      U     "G299M".A_3235_MXZ11.StHN   // Louver Air Heater Kilningbox 2
//MW 2010.04.29      U     "G273M".A_3136_MXZ11.StHN   // Recycling Air Flap Kilningbox 1
// Luft-Austritt
//MW 2010.04.29      U     "G273M".A_3135_MXZ11.StHN   // Recycling Air Flap Kilningbox 1
//MW 2010.04.29      UN    "G273M".A_3136_MXZ11.StLN   // Recycling Air Flap Kilningbox 1
//MW 2010.04.29      UN    "G299M".A_3236_MXZ11.StLN   // Recycling Air Flap Kilningbox 2
// 100% Umluft-Betrieb
//MW 2010.04.29      U     "G273M".A_3135_MXZ11.StHN   // Recycling Air Flap Kilningbox 1
//MW 2010.04.29      O     "G273M".A_3136_MXZ11.StHN   // Recycling Air Flap Kilningbox 1
//MW 2010.04.29      O     "G299M".A_3236_MXZ11.StHN   // Recycling Air Flap Kilningbox 2
//MW 2010.04.13
NETWORK
TITLE = Interlocking Next
      A     DIX [AR2,P#15.2];
      A     DIX [AR2,P#18.4];
      AN    DIX [AR2,P#19.6];
      =     #tmpCmdNext;
NETWORK
TITLE = Interlocking Local / HWStop
      A     DB50.DBX 32.3;
      =     #tmpHWStop;
      A     DIX [AR2,P#16.0];
      O     #tmpHWStop;
      =     #tmpLocal;
NETWORK
TITLE = Interlocking Start Warning
      NOP   0;
//- Restart after fault --
      A     DIX [AR2,P#15.3];
      A     DIX [AR2,P#19.2];
      S     DB100.DBX 126.4;
//- Run Timer --
      OPN   "G271M";
      CALL  FB 100 , DB 100 (
           DIX 0.0                  := FALSE,
           DIW 2                    := 10,
           DIX 4.0                  := DBX [AR2,P#18.0],
           DIX 4.1                  := #tmpLocal,
           DIX 4.2                  := DBX [AR2,P#19.1],
           DIX 4.3                  := #tmpCmdNext,
           DIX 6.0                  := #tmpCmdNext,
           DIX 6.1                  := DBX [AR2,P#19.3]);
//- Store Startwarning done  --
//- Reset Autostart --
      A     DB100.DBX 236.1;
      FN    DIX [AR2,P#58.7];
      A     DIX [AR2,P#19.2];
      R     DIX [AR2,P#18.4];
NETWORK
TITLE = =A-3125-KCU04AI1 : VIBRATION MONITOR FAN 1 CHANNEL 1
//Alarm Level = 10.00mm/sec
//Trip Level = 11.20mm/sec
//MW 2010.04.09
      NOP   0;
//-InLocal---
      A     #tmpLocal;
      O     DB922.DBX 1569.0;	// emergency regime without fan 1
      =     DIX [AR2,P#63.4];
//-Monitoring--- 
      CLR;
      =     DIX [AR2,P#62.0];
      CLR;
      =     DIX [AR2,P#62.1];
      CLR;
      =     DIX [AR2,P#62.2];
      SET;
      =     DIX [AR2,P#62.3];
      SET;
      =     DIX [AR2,P#62.4];
// 
//-Read inputs---
      L     PIW 954;
      L     0;
      <I;
      JC    v003;
      TAK;
v003: T     DIW [AR2,P#66.0];
      A     DB50.DBX 32.3;
      =     DIX [AR2,P#63.0];
      A     DB51.DBX 11.3;
      =     DIX [AR2,P#63.1];
// 
//-Set Parameters---
// --> Erläuterung
      L     L#2540;	// 20mA = 25.40mm/sec       
      T     DB371.DBD 90;
      L     L#10000;	// OutValuePc=OutValueUnits
      T     DB371.DBD 94;
      L     L#-1;	// -0.01mm/sec
      T     DB371.DBD 98;
      L     L#0;	// 0.00mm/sec
      T     DB371.DBD 102;
      L     L#1000;	// 10.00mm/sec
      T     DB371.DBD 106;
      L     L#1120;	// 11.20mm/sec
      T     DB371.DBD 110;
      SET;
      =     DB371.DBX 84.6;
      =     DB371.DBX 84.7;
      =     DB371.DBX 85.0;
      =     DB371.DBX 85.1;
      =     DB371.DBX 85.6;
      =     DB371.DBX 85.7;
      CLR;
      =     DB371.DBX 85.2;
// 
//-Call object control---
      BLD   14;
// 
//-Write outputs---  
      =     L 10.0;
      L     DINO;
      T     LW 8;
      CDB;
      OPN   DI [LW 8];
      TAR2  LD 4;
      +AR2  P#60.0;
      UC    FB 19;
      LAR2  LD 4;
      CDB;
      BLD   15;
NETWORK
TITLE = =A-3125-KCU04AI2 : VIBRATION MONITOR FAN 1 CHANNEL 2
//Alarm Level = 10.00mm/sec
//Trip Level = 11.20mm/sec
//MW 2010.04.09
      NOP   0;
//-InLocal---
      A     #tmpLocal;
      O     DB922.DBX 1569.0;	// emergency regime without fan 1
      =     DIX [AR2,P#151.4];
//-Monitoring--- 
      CLR;
      =     DIX [AR2,P#150.0];
      CLR;
      =     DIX [AR2,P#150.1];
      CLR;
      =     DIX [AR2,P#150.2];
      SET;
      =     DIX [AR2,P#150.3];
      SET;
      =     DIX [AR2,P#150.4];
// 
//-Read inputs---
      L     PIW 952;
      L     0;
      <I;
      JC    v004;
      TAK;
v004: T     DIW [AR2,P#154.0];
      A     DB50.DBX 32.3;
      =     DIX [AR2,P#151.0];
      A     DB51.DBX 11.3;
      =     DIX [AR2,P#151.1];
// 
//-Set Parameters---
// --> Erläuterung
      L     L#2540;	// 20mA = 25.40mm/sec       
      T     DB371.DBD 178;
      L     L#10000;	// OutValuePc=OutValueUnits
      T     DB371.DBD 182;
      L     L#-1;	// -0.01mm/sec
      T     DB371.DBD 186;
      L     L#0;	// 0.00mm/sec
      T     DB371.DBD 190;
      L     L#1000;	// 10.00mm/sec
      T     DB371.DBD 194;
      L     L#1120;	// 11.20mm/sec
      T     DB371.DBD 198;
      SET;
      =     DB371.DBX 172.6;
      =     DB371.DBX 172.7;
      =     DB371.DBX 173.0;
      =     DB371.DBX 173.1;
      =     DB371.DBX 173.6;
      =     DB371.DBX 173.7;
      CLR;
      =     DB371.DBX 173.2;
// 
//-Call object control---
      BLD   14;
// 
//-Write outputs---
      =     L 10.0;
      L     DINO;
      T     LW 8;
      CDB;
      OPN   DI [LW 8];
      TAR2  LD 4;
      +AR2  P#148.0;
      UC    FB 19;
      LAR2  LD 4;
      CDB;
      BLD   15;
NETWORK
TITLE = =A-3125-BTE05 : TEMPERATURE BEARING TEMPERATUR SENSOR
//Alarm Level = 100.00°C    
//Trip Level = 110.00°C
//MW 2010.04.09
      NOP   0;
//-InLocal---
      A     #tmpLocal;
      O     DB922.DBX 1569.0;	// emergency regime without fan 1
      =     DIX [AR2,P#239.4];
//-Monitoring--- 
      CLR;
      =     DIX [AR2,P#238.0];
      CLR;
      =     DIX [AR2,P#238.1];
      CLR;
      =     DIX [AR2,P#238.2];
      SET;
      =     DIX [AR2,P#238.3];
      SET;
      =     DIX [AR2,P#238.4];
// 
//-Read inputs---
      L     PIW 928;
      T     DIW [AR2,P#242.0];
      A     DB50.DBX 32.3;
      =     DIX [AR2,P#239.0];
      A     DB51.DBX 11.3;
      =     DIX [AR2,P#239.1];
//To Block Problems with Sensor
      L     600;
      T     DB371.DBW 296;
      T     DB371.DBW 298;
// 
//-Set Parameters---
// --> Erläuterung
      L     L#27648;	// Temperature direkt      
      T     DB371.DBD 266;
      L     L#10000;	// OutValuePc=OutValueUnits
      T     DB371.DBD 270;
      L     L#0;	// 0.00°C
      T     DB371.DBD 274;
      L     L#100;	// 1.00°C
      T     DB371.DBD 278;
      L     L#10000;	// 100.00°C
      T     DB371.DBD 282;
      L     L#11000;	// 110.00°C
      T     DB371.DBD 286;
      SET;
      =     DB371.DBX 260.6;
      =     DB371.DBX 260.7;
      =     DB371.DBX 261.0;
      =     DB371.DBX 261.1;
      =     DB371.DBX 261.6;
      =     DB371.DBX 261.7;
      CLR;
      =     DB371.DBX 261.2;
// 
//-Call object control---
      BLD   14;
// 
//-Write outputs---      
      =     L 10.0;
      L     DINO;
      T     LW 8;
      CDB;
      OPN   DI [LW 8];
      TAR2  LD 4;
      +AR2  P#236.0;
      UC    FB 19;
      LAR2  LD 4;
      CDB;
      BLD   15;
NETWORK
TITLE = =A-3125-BTE06 : TEMPERATURE BEARING TEMPERATUR SENSOR
//Alarm Level = 100.00°C    
//Trip Level = 110.00°C
//MW 2010.04.09
      NOP   0;
//-InLocal---
      A     #tmpLocal;
      O     DB922.DBX 1569.0;	// emergency regime without fan 1
      =     DIX [AR2,P#327.4];
//-Monitoring--- 
      CLR;
      =     DIX [AR2,P#326.0];
      CLR;
      =     DIX [AR2,P#326.1];
      CLR;
      =     DIX [AR2,P#326.2];
      SET;
      =     DIX [AR2,P#326.3];
      SET;
      =     DIX [AR2,P#326.4];
// 
//-Read inputs---
      L     PIW 930;
      T     DIW [AR2,P#330.0];
      A     DB50.DBX 32.3;
      =     DIX [AR2,P#327.0];
      A     DB51.DBX 11.3;
      =     DIX [AR2,P#327.1];
//To Block Problems with Sensor
      L     600;
      T     DB371.DBW 384;
      T     DB371.DBW 386;
// 
//-Set Parameters---
// --> Erläuterung
      L     L#27648;	// Temperature direkt      
      T     DB371.DBD 354;
      L     L#10000;	// OutValuePc=OutValueUnits
      T     DB371.DBD 358;
      L     L#0;	// 0.00°C
      T     DB371.DBD 362;
      L     L#100;	// 1.00°C
      T     DB371.DBD 366;
      L     L#10000;	// 100.00°C
      T     DB371.DBD 370;
      L     L#11000;	// 110.00°C
      T     DB371.DBD 374;
      SET;
      =     DB371.DBX 348.6;
      =     DB371.DBX 348.7;
      =     DB371.DBX 349.0;
      =     DB371.DBX 349.1;
      =     DB371.DBX 349.6;
      =     DB371.DBX 349.7;
      CLR;
      =     DB371.DBX 349.2;
// 
//-Call object control---
      BLD   14;
// 
//-Write outputs---
      =     L 10.0;
      L     DINO;
      T     LW 8;
      CDB;
      OPN   DI [LW 8];
      TAR2  LD 4;
      +AR2  P#324.0;
      UC    FB 19;
      LAR2  LD 4;
      CDB;
      BLD   15;
NETWORK
TITLE = =A-3125-MXZ01MA : FAN 1
      NOP   0;
//-InLocal---
      A     #tmpLocal;
      O     DB922.DBX 1569.0;	// emergency regime without fan 1
      =     DIX [AR2,P#415.4];
//-Interlocking---
      AN    DB922.DBX 1569.0;	// emergency regime without fan 1
      A(;
      AN    DIX [AR2,P#1411.4];
      O     DB922.DBX 1569.1;	// emergency regime without fan 2
      );
      A(;
      A     DIX [AR2,P#15.5];
      A     DIX [AR2,P#14.5];
      ON    DIX [AR2,P#15.5];
      );
      AN    DIX [AR2,P#65.7];	// Vibrationswächter 1
      AN    DIX [AR2,P#153.7];	// Vibrationswächter 2
      AN    DIX [AR2,P#241.7];	// Lager Temperatur 1
      AN    DIX [AR2,P#329.7];	// Lager Temperatur 2
      AN    DB376.DBX 65.4;	// Differenzdruck hinter dem Waermetauscher
      A     DIX [AR2,P#18.0];
      =     DIX [AR2,P#414.1];
      A     #tmpCmdNext;
//      U     "MAL1S032Par".Par.FlagProcess2.Schaltp_5
      S     DIX [AR2,P#415.2];
      A     DIX [AR2,P#19.7];
      =     DIX [AR2,P#415.7];
// 
//=Values and commands of elements===
//-=A-3125-KCU04---
//      CLR
//      S     #A_3125_MXZ01MA.A_3125_KCU04.CmdRunTimeOutTime
//-=A-3125-MXZ01_SM---
//      CLR
//      S     #A_3125_MXZ01MA.A_3125_MXZ01_SM.CmdRunTimeOutTime
// 
//-Read inputs of elements---
//KR04022010 kein speed monitor vorhanden---->
      O     DB371.DBX 417.1;
      O     DB371.DBX 417.2;
      =     DB371.DBX 460.6;
//<----
      A     I 926.6;
      =     DIX [AR2,P#426.6];
      A     DB50.DBX 32.3;
      =     DIX [AR2,P#428.0];
      A     DB51.DBX 11.4;
      =     DIX [AR2,P#428.1];
      A     DB50.DBX 32.3;
      =     DIX [AR2,P#462.0];
//MW 2010.04.09
      A     DIX [AR2,P#664.4];
      O     DB50.DBX 33.0;
      A     DIX [AR2,P#632.6];
      =     DIX [AR2,P#630.6];
      A     DB50.DBX 32.3;
      =     DIX [AR2,P#632.0];
// MW 2010.04.09 - Überwachung Profibus-Kommunikation
      A     DB51.DBX 11.5;	// FU
      =     DIX [AR2,P#632.1];
// 
//-Set Parameters---
// 
//-Call object control---
      BLD   14;
// 
//-Write outputs---
      =     L 10.0;
      L     DINO;
      T     LW 8;
      CDB;
      OPN   DI [LW 8];
      TAR2  LD 4;
      +AR2  P#412.0;
      UC    "A_3125_MXZ01MA_Code";
      LAR2  LD 4;
      CDB;
      BLD   15;
NETWORK
TITLE = =A-3125-TSC01_COM : FAN 1 FU KOMMUNIKATION
      NOP   0;
      A     DIX [AR2,P#632.6];
      =     DIX [AR2,P#664.1];
//      U     #A_3125_MXZ01MA.A_3125_MXZ01.OutpRunRev
      CLR;
      =     DIX [AR2,P#664.0];
      A     DIX [AR2,P#15.3];
      O     DIX [AR2,P#428.6];
      S     DIX [AR2,P#664.2];
// 
//-Read inputs---
// 
//-Set Parameters---
// 
//-Call object control---
      BLD   14;
// 
//-Write outputs---
      =     L 10.0;
      L     DINO;
      T     LW 8;
      CDB;
      OPN   DI [LW 8];
      TAR2  LD 4;
      +AR2  P#662.0;
      UC    FB 1816;
      LAR2  LD 4;
      CDB;
      BLD   15;
NETWORK
TITLE = =A-3125-TSC01_AC : ACT. CURRENT FAN 1 FU 
//20000Dez=100,0%=720,0A
//Analog Input 20mA=27648Dez=995,3A
      NOP   0;
//-InLocal---
      A     #tmpLocal;
      O     DB922.DBX 1569.0;	// emergency regime without fan 1
      =     DIX [AR2,P#705.4];
//-Monitoring--- 
      SET;
      =     DIX [AR2,P#704.0];
      CLR;
      =     DIX [AR2,P#704.1];
      CLR;
      =     DIX [AR2,P#704.2];
      CLR;
      =     DIX [AR2,P#704.3];
      CLR;
      =     DIX [AR2,P#704.4];
// 
//-Read inputs---
//MW 2010.04.09      L     #A_3125_TSC01_COM.Output.SetpointValue01
//MW 2010.04.09      ITD   
//MW 2010.04.09      DTR   
//MW 2010.04.09      ABS   
//MW 2010.04.09      RND   
      L     DIW [AR2,P#672.0];
      T     DIW [AR2,P#708.0];
      A     DB50.DBX 32.3;
      =     DIX [AR2,P#705.0];
// 
//-Set Parameters---
//MW 2010.04.09
      L     L#9953;	// Stromwert bei 27648Dez
      T     DB371.DBD 732;
      L     L#10000;	// OutValuePc=OutValueUnits
      T     DB371.DBD 736;
      L     L#0;	// 0.0A
      T     DB371.DBD 740;
      L     L#4000;	// 40.0A
      T     DB371.DBD 744;
      L     L#7200;	// 720.0A=100.0%
      T     DB371.DBD 748;
      L     L#9360;	// 936.0A=130.0%
      T     DB371.DBD 752;
// 
//-Call object control---
      BLD   14;
// 
//-Write outputs---
      =     L 10.0;
      L     DINO;
      T     LW 8;
      CDB;
      OPN   DI [LW 8];
      TAR2  LD 4;
      +AR2  P#702.0;
      UC    FB 19;
      LAR2  LD 4;
      CDB;
      BLD   15;
NETWORK
TITLE = =A-3125-TSC01_AF : ACT. FREQUENCY FAN 1 FU 
      NOP   0;
//-InLocal---
      A     #tmpLocal;
      O     DB922.DBX 1569.0;	// emergency regime without fan 1
      =     DIX [AR2,P#793.4];
//-Monitoring--- 
      SET;
      =     DIX [AR2,P#792.0];
      CLR;
      =     DIX [AR2,P#792.1];
      CLR;
      =     DIX [AR2,P#792.2];
      CLR;
      =     DIX [AR2,P#792.3];
      CLR;
      =     DIX [AR2,P#792.4];
// 
//-Read inputs---
//MW 2010.04.09      L     #A_3125_TSC01_COM.Output.SetpointValue01
//MW 2010.04.09      ITD   
//MW 2010.04.09      DTR   
//MW 2010.04.09      ABS   
//MW 2010.04.09      RND   
      L     DIW [AR2,P#662.0];	// Umgerechnet in FU-FB
      L     10000;	//BRT - Testsystem
      T     DIW [AR2,P#796.0];
      A     DB50.DBX 32.3;
      =     DIX [AR2,P#793.0];
// 
//-Set Parameters---
//MW 2010.04.09
      L     L#27648;	// InpValue=Drehzahl direkt   
      T     DB371.DBD 820;
      L     L#10000;	// OutValuePc=OutValueUnits
      T     DB371.DBD 824;
      L     L#4000;	// 40.00% ist untere Grenze
      T     DB371.DBD 828;
      L     L#4100;	// 41.00%
      T     DB371.DBD 832;
      L     L#8000;	// 80.00%
      T     DB371.DBD 836;
      L     L#10100;	// 101.00%
      T     DB371.DBD 840;
// 
//-Call object control---
      BLD   14;
// 
//-Write outputs---
      =     L 10.0;
      L     DINO;
      T     LW 8;
      CDB;
      OPN   DI [LW 8];
      TAR2  LD 4;
      +AR2  P#790.0;
      UC    FB 19;
      LAR2  LD 4;
      CDB;
      BLD   15;
NETWORK
TITLE = =A-3125-TSC01_AT : ACT. TORQUE FAN 1 FU 
      NOP   0;
//-InLocal---
      A     #tmpLocal;
      O     DB922.DBX 1569.0;	// emergency regime without fan 1
      =     DIX [AR2,P#881.4];
//-Monitoring--- 
      CLR;
      =     DIX [AR2,P#880.0];
      CLR;
      =     DIX [AR2,P#880.1];
      CLR;
      =     DIX [AR2,P#880.2];
      CLR;
      =     DIX [AR2,P#880.3];
      CLR;
      =     DIX [AR2,P#880.4];
// 
//-Read inputs---
//MW 2010.04.09      L     #A_3125_TSC01_COM.Output.SetpointValue01
//MW 2010.04.09      ITD   
//MW 2010.04.09      DTR   
//MW 2010.04.09      ABS   
//MW 2010.04.09      RND   
      L     DIW [AR2,P#676.0];
      T     DIW [AR2,P#884.0];
      A     DB50.DBX 32.3;
      =     DIX [AR2,P#881.0];
// 
//-Set Parameters---
// 
//-Call object control---
      BLD   14;
// 
//-Write outputs---
      =     L 10.0;
      L     DINO;
      T     LW 8;
      CDB;
      OPN   DI [LW 8];
      TAR2  LD 4;
      +AR2  P#878.0;
      UC    FB 19;
      LAR2  LD 4;
      CDB;
      BLD   15;
NETWORK
TITLE = =A-3125-TSC01_AP : ACT. POWER FAN 1 FU 
      NOP   0;
//-InLocal---
      A     #tmpLocal;
      O     DB922.DBX 1569.0;	// emergency regime without fan 1
      =     DIX [AR2,P#969.4];
//-Monitoring--- 
      CLR;
      =     DIX [AR2,P#968.0];
      CLR;
      =     DIX [AR2,P#968.1];
      CLR;
      =     DIX [AR2,P#968.2];
      CLR;
      =     DIX [AR2,P#968.3];
      CLR;
      =     DIX [AR2,P#968.4];
// 
//-Read inputs---
//MW 2010.04.09      L     #A_3125_TSC01_COM.Output.SetpointValue01
//MW 2010.04.09      ITD   
//MW 2010.04.09      DTR   
//MW 2010.04.09      ABS   
//MW 2010.04.09      RND   
      L     DIW [AR2,P#674.0];
      T     DIW [AR2,P#972.0];
      A     DB50.DBX 32.3;
      =     DIX [AR2,P#969.0];
// 
//-Set Parameters---
// 
//-Call object control---
      BLD   14;
// 
//-Write outputs---
      =     L 10.0;
      L     DINO;
      T     LW 8;
      CDB;
      OPN   DI [LW 8];
      TAR2  LD 4;
      +AR2  P#966.0;
      UC    FB 19;
      LAR2  LD 4;
      CDB;
      BLD   15;
NETWORK
TITLE = =A-3126-KCU04AI1 : VIBRATION MONITOR FAN 2 CHANNEL 1
//Alarm Level = 10.00mm/sec
//Trip Level = 11.20mm/sec
//MW 2010.04.09
      NOP   0;
//-InLocal---
      A     #tmpLocal;
      O     DB922.DBX 1569.1;	// emergency regime without fan 2
      =     DIX [AR2,P#1057.4];
//-Monitoring--- 
      CLR;
      =     DIX [AR2,P#1056.0];
      CLR;
      =     DIX [AR2,P#1056.1];
      CLR;
      =     DIX [AR2,P#1056.2];
      SET;
      =     DIX [AR2,P#1056.3];
      SET;
      =     DIX [AR2,P#1056.4];
// 
//-Read inputs---
      L     PIW 958;
      L     0;
      <I;
      JC    v013;
      TAK;
v013: T     DIW [AR2,P#1060.0];
      A     DB50.DBX 32.3;
      =     DIX [AR2,P#1057.0];
      A     DB51.DBX 11.3;
      =     DIX [AR2,P#1057.1];
// 
//-Set Parameters---
// --> Erläuterung
      L     L#2540;	// 20mA = 25.40mm/sec       
      T     DB371.DBD 1084;
      L     L#10000;	// OutValuePc=OutValueUnits
      T     DB371.DBD 1088;
      L     L#-1;	// -0.01mm/sec
      T     DB371.DBD 1092;
      L     L#0;	// 0.00mm/sec
      T     DB371.DBD 1096;
      L     L#1000;	// 10.00mm/sec
      T     DB371.DBD 1100;
      L     L#1120;	// 11.20mm/sec
      T     DB371.DBD 1104;
      SET;
      =     DB371.DBX 1078.6;
      =     DB371.DBX 1078.7;
      =     DB371.DBX 1079.0;
      =     DB371.DBX 1079.1;
      =     DB371.DBX 1079.6;
      =     DB371.DBX 1079.7;
      CLR;
      =     DB371.DBX 1079.2;
// 
//-Call object control---
      BLD   14;
// 
//-Write outputs---
      =     L 10.0;
      L     DINO;
      T     LW 8;
      CDB;
      OPN   DI [LW 8];
      TAR2  LD 4;
      +AR2  P#1054.0;
      UC    FB 19;
      LAR2  LD 4;
      CDB;
      BLD   15;
NETWORK
TITLE = =A-3126-KCU04AI2 : VIBRATION MONITOR FAN 2 CHANNEL 2
//Alarm Level = 10.00mm/sec
//Trip Level = 11.20mm/sec
//MW 2010.04.09
      NOP   0;
//-InLocal---
      A     #tmpLocal;
      O     DB922.DBX 1569.1;	// emergency regime without fan 2
      =     DIX [AR2,P#1145.4];
//-Monitoring--- 
      CLR;
      =     DIX [AR2,P#1144.0];
      CLR;
      =     DIX [AR2,P#1144.1];
      CLR;
      =     DIX [AR2,P#1144.2];
      CLR;
      =     DIX [AR2,P#1144.3];
      SET;
      =     DIX [AR2,P#1144.4];
// 
//-Read inputs---
      L     PIW 956;
      L     0;
      <I;
      JC    v014;
      TAK;
v014: T     DIW [AR2,P#1148.0];
      A     DB50.DBX 32.3;
      =     DIX [AR2,P#1145.0];
      A     DB51.DBX 11.3;
      =     DIX [AR2,P#1145.1];
// 
//-Set Parameters---
// --> Erläuterung
      L     L#2540;	// 20mA = 25.40mm/sec       
      T     DB371.DBD 1172;
      L     L#10000;	// OutValuePc=OutValueUnits
      T     DB371.DBD 1176;
      L     L#-1;	// -0.01mm/sec
      T     DB371.DBD 1180;
      L     L#0;	// 0.00mm/sec
      T     DB371.DBD 1184;
      L     L#1000;	// 10.00mm/sec
      T     DB371.DBD 1188;
      L     L#1120;	// 11.20mm/sec
      T     DB371.DBD 1192;
      SET;
      =     DB371.DBX 1166.6;
      =     DB371.DBX 1166.7;
      =     DB371.DBX 1167.0;
      =     DB371.DBX 1167.1;
      =     DB371.DBX 1167.6;
      =     DB371.DBX 1167.7;
      CLR;
      =     DB371.DBX 1167.2;
// 
//-Call object control---
      BLD   14;
// 
//-Write outputs---
      =     L 10.0;
      L     DINO;
      T     LW 8;
      CDB;
      OPN   DI [LW 8];
      TAR2  LD 4;
      +AR2  P#1142.0;
      UC    FB 19;
      LAR2  LD 4;
      CDB;
      BLD   15;
NETWORK
TITLE = =A-3126-BTE05 : TEMPERATURE BEARING TEMPERATUR SENSOR
//Alarm Level = 100.00°C    
//Trip Level = 110.00°C
//MW 2010.04.09
      NOP   0;
//-InLocal---
      A     #tmpLocal;
      O     DB922.DBX 1569.1;	// emergency regime without fan 2
      =     DIX [AR2,P#1233.4];
//-Monitoring--- 
      CLR;
      =     DIX [AR2,P#1232.0];
      CLR;
      =     DIX [AR2,P#1232.1];
      CLR;
      =     DIX [AR2,P#1232.2];
      SET;	// CLR
      =     DIX [AR2,P#1232.3];
      SET;
      =     DIX [AR2,P#1232.4];
// 
//-Read inputs---
      L     PIW 932;
      T     DIW [AR2,P#1236.0];
      A     DB50.DBX 32.3;
      =     DIX [AR2,P#1233.0];
      A     DB51.DBX 11.3;
      =     DIX [AR2,P#1233.1];
// 
//To Block Problems with Sensor
      L     600;
      T     DB371.DBW 1290;
      T     DB371.DBW 1292;
// 
//-Set Parameters---
// --> Erläuterung
      L     L#27648;	// Temperature direkt      
      T     DB371.DBD 1260;
      L     L#10000;	// OutValuePc=OutValueUnits
      T     DB371.DBD 1264;
      L     L#0;	// 0.00°C
      T     DB371.DBD 1268;
      L     L#100;	// 1.00°C
      T     DB371.DBD 1272;
      L     L#10000;	// 100.00°C
      T     DB371.DBD 1276;
      L     L#11000;	// 110.00°C
      T     DB371.DBD 1280;
      SET;
      =     DB371.DBX 1254.6;
      =     DB371.DBX 1254.7;
      =     DB371.DBX 1255.0;
      =     DB371.DBX 1255.1;
      =     DB371.DBX 1255.6;
      =     DB371.DBX 1255.7;
      CLR;
      =     DB371.DBX 1255.2;
// 
//-Call object control---
      BLD   14;
// 
//-Write outputs---
      =     L 10.0;
      L     DINO;
      T     LW 8;
      CDB;
      OPN   DI [LW 8];
      TAR2  LD 4;
      +AR2  P#1230.0;
      UC    FB 19;
      LAR2  LD 4;
      CDB;
      BLD   15;
NETWORK
TITLE = =A-3126-BTE06 : TEMPERATURE BEARING TEMPERATUR SENSOR
//Alarm Level = 100.00°C    
//Trip Level = 110.00°C
//MW 2010.04.09
      NOP   0;
//-InLocal---
      A     #tmpLocal;
      O     DB922.DBX 1569.1;	// emergency regime without fan 2
      =     DIX [AR2,P#1321.4];
//-Monitoring--- 
      CLR;
      =     DIX [AR2,P#1320.0];
      CLR;
      =     DIX [AR2,P#1320.1];
      CLR;
      =     DIX [AR2,P#1320.2];
      SET;	//CLR   
      =     DIX [AR2,P#1320.3];
      SET;
      =     DIX [AR2,P#1320.4];
// 
//-Read inputs---
      L     PIW 934;
      T     DIW [AR2,P#1324.0];
      A     DB50.DBX 32.3;
      =     DIX [AR2,P#1321.0];
      A     DB51.DBX 11.3;
      =     DIX [AR2,P#1321.1];
// 
//To Block Problems with Sensor
      L     600;
      T     DB371.DBW 1378;
      T     DB371.DBW 1380;
// 
//-Set Parameters---
// --> Erläuterung
      L     L#27648;	// Temperature direkt      
      T     DB371.DBD 1348;
      L     L#10000;	// OutValuePc=OutValueUnits
      T     DB371.DBD 1352;
      L     L#0;	// 0.00°C
      T     DB371.DBD 1356;
      L     L#100;	// 1.00°C
      T     DB371.DBD 1360;
      L     L#10000;	// 100.00°C
      T     DB371.DBD 1364;
      L     L#11000;	// 110.00°C
      T     DB371.DBD 1368;
      SET;
      =     DB371.DBX 1342.6;
      =     DB371.DBX 1342.7;
      =     DB371.DBX 1343.0;
      =     DB371.DBX 1343.1;
      =     DB371.DBX 1343.6;
      =     DB371.DBX 1343.7;
      CLR;
      =     DB371.DBX 1343.2;
// 
//-Call object control---
      BLD   14;
// 
//-Write outputs---
      =     L 10.0;
      L     DINO;
      T     LW 8;
      CDB;
      OPN   DI [LW 8];
      TAR2  LD 4;
      +AR2  P#1318.0;
      UC    FB 19;
      LAR2  LD 4;
      CDB;
      BLD   15;
NETWORK
TITLE = =A-3126-MXZ01MA : FAN 2
      NOP   0;
//-InLocal---
      A     #tmpLocal;
      O     DB922.DBX 1569.1;	// emergency regime without fan 2
      =     DIX [AR2,P#1409.4];
//-Interlocking---
//MW 2010.04.09
      AN    DB922.DBX 1569.1;	// emergency regime without fan 2
      A(;
      AN    DIX [AR2,P#417.4];
      O     DB922.DBX 1569.0;	// emergency regime without fan 1
      );
      A(;
      A     DIX [AR2,P#15.5];
      A     DIX [AR2,P#14.5];
      ON    DIX [AR2,P#15.5];
      );
      AN    DIX [AR2,P#1059.7];	// Vibrationswächter 1
      AN    DIX [AR2,P#1147.7];	// Vibrationswächter 2
      AN    DIX [AR2,P#1235.7];	// Lager Temperatur 1
      AN    DIX [AR2,P#1323.7];	// Lager Temperatur 2
      AN    DB376.DBX 65.4;	// Differenzdruck hinter dem Waermetauscher
      A     DIX [AR2,P#18.0];
      =     DIX [AR2,P#1408.1];
      A     #tmpCmdNext;
//      U     "MAL1S032Par".Par.FlagProcess2.Schaltp_5
      S     DIX [AR2,P#1409.2];
      A     DIX [AR2,P#19.7];
      =     DIX [AR2,P#1409.7];
// 
//=Values and commands of elements===
//-=A-3126-KCU04---
//      CLR
//      S     #A_3126_MXZ01MA.A_3126_KCU04.CmdRunTimeOutTime
//-=A-3126-MXZ01_SM---
//      CLR
//      S     #A_3126_MXZ01MA.A_3126_MXZ01_SM.CmdRunTimeOutTime
// 
//-Read inputs of elements---
//KR04022010 kein speed monitor vorhanden---->
      O     DB371.DBX 1411.1;
      O     DB371.DBX 1411.2;
      =     DB371.DBX 1454.6;
//<----
      A     I 926.7;
      =     DIX [AR2,P#1420.6];
      A     DB50.DBX 32.3;
      =     DIX [AR2,P#1422.0];
      A     DB51.DBX 11.4;
      =     DIX [AR2,P#1422.1];
      A     DB50.DBX 32.3;
      =     DIX [AR2,P#1456.0];
//MW 2010.04.09
      A     DIX [AR2,P#1658.4];
      O     DB50.DBX 33.0;
      A     DIX [AR2,P#1626.6];
      =     DIX [AR2,P#1624.6];
      A     DB50.DBX 32.3;
      =     DIX [AR2,P#1626.0];
// MW 2010.04.09 - Überwachung Profibus-Kommunikation
      A     DB51.DBX 11.6;	// FU
      =     DIX [AR2,P#1626.1];
// 
//-Set Parameters---
// 
//-Call object control---
      BLD   14;
// 
//-Write outputs---
      =     L 10.0;
      L     DINO;
      T     LW 8;
      CDB;
      OPN   DI [LW 8];
      TAR2  LD 4;
      +AR2  P#1406.0;
      UC    "A_3126_MXZ01MA_Code";
      LAR2  LD 4;
      CDB;
      BLD   15;
NETWORK
TITLE = =A-3126-TSC01_COM : FAN 2 FU KOMMUNIKATION
      NOP   0;
      A     DIX [AR2,P#1626.6];
      =     DIX [AR2,P#1658.1];
//      U     #A_3126_MXZ01MA.A_3126_MXZ01.OutpRunRev
      CLR;
      =     DIX [AR2,P#1658.0];
      A     DIX [AR2,P#15.3];
      O     DIX [AR2,P#1422.6];
      S     DIX [AR2,P#1658.2];
// 
//-Read inputs---
// 
//-Set Parameters---
// 
//-Call object control---
      BLD   14;
// 
//-Write outputs---
      =     L 10.0;
      L     DINO;
      T     LW 8;
      CDB;
      OPN   DI [LW 8];
      TAR2  LD 4;
      +AR2  P#1656.0;
      UC    FB 1816;
      LAR2  LD 4;
      CDB;
      BLD   15;
NETWORK
TITLE = =A-3126-TSC01_AC : ACT. CURRENT FAN 2 FU 
//20000Dez=100,0%=720,0A
//Analog Input 20mA=27648Dez=995,3A
      NOP   0;
//-InLocal---
      A     #tmpLocal;
      O     DB922.DBX 1569.1;	// emergency regime without fan 2
      =     DIX [AR2,P#1699.4];
//-Monitoring--- 
      SET;
      =     DIX [AR2,P#1698.0];
      CLR;
      =     DIX [AR2,P#1698.1];
      CLR;
      =     DIX [AR2,P#1698.2];
      CLR;
      =     DIX [AR2,P#1698.3];
      CLR;	//SET   
      =     DIX [AR2,P#1698.4];
// 
//-Read inputs---
//MW 2010.04.09      L     #A_3126_TSC01_COM.Output.SetpointValue01
//MW 2010.04.09      ITD   
//MW 2010.04.09      DTR   
//MW 2010.04.09      ABS   
//MW 2010.04.09      RND   
      L     DIW [AR2,P#1666.0];
      T     DIW [AR2,P#1702.0];
      A     DB50.DBX 32.3;
      =     DIX [AR2,P#1699.0];
// 
//-Set Parameters---
//MW 2010.04.09
      L     L#9953;	// Stromwert bei 27648Dez
      T     DB371.DBD 1726;
      L     L#10000;	// OutValuePc=OutValueUnits
      T     DB371.DBD 1730;
      L     L#0;	// 0.0A
      T     DB371.DBD 1734;
      L     L#4000;	// 40.0A
      T     DB371.DBD 1738;
      L     L#7200;	// 720.0A=100.0%
      T     DB371.DBD 1742;
      L     L#9360;	// 936.0A=130.0%
      T     DB371.DBD 1746;
// 
//-Call object control---
      BLD   14;
// 
//-Write outputs---
      =     L 10.0;
      L     DINO;
      T     LW 8;
      CDB;
      OPN   DI [LW 8];
      TAR2  LD 4;
      +AR2  P#1696.0;
      UC    FB 19;
      LAR2  LD 4;
      CDB;
      BLD   15;
NETWORK
TITLE = =A-3126-TSC01_AF : ACT. FREQUENCY FAN 2 FU 
      NOP   0;
//-InLocal---
      A     #tmpLocal;
      O     DB922.DBX 1569.1;	// emergency regime without fan 2
      =     DIX [AR2,P#1787.4];
//-Monitoring--- 
      SET;
      =     DIX [AR2,P#1786.0];
      CLR;
      =     DIX [AR2,P#1786.1];
      CLR;
      =     DIX [AR2,P#1786.2];
      CLR;
      =     DIX [AR2,P#1786.3];
      CLR;
      =     DIX [AR2,P#1786.4];
// 
//-Read inputs---
//MW 2010.04.09      L     #A_3126_TSC01_COM.Output.SetpointValue01
//MW 2010.04.09      ITD   
//MW 2010.04.09      DTR   
//MW 2010.04.09      ABS   
//MW 2010.04.09      RND   
      L     DIW [AR2,P#1656.0];	// Umgerechnet in FU-FB
      L     10000;	//BRT - Testsystem
      T     DIW [AR2,P#1790.0];
      A     DB50.DBX 32.3;
      =     DIX [AR2,P#1787.0];
// 
//-Set Parameters---
//MW 2010.04.09
      L     L#27648;	// InpValue=Drehzahl direkt   
      T     DB371.DBD 1814;
      L     L#10000;	// OutValuePc=OutValueUnits
      T     DB371.DBD 1818;
      L     L#4000;	// 40.00% ist untere Grenze
      T     DB371.DBD 1822;
      L     L#4100;	// 41.00%
      T     DB371.DBD 1826;
      L     L#8000;	// 80.00%
      T     DB371.DBD 1830;
      L     L#10100;	// 101.00%
      T     DB371.DBD 1834;
// 
//-Call object control---
      BLD   14;
// 
//-Write outputs---
      =     L 10.0;
      L     DINO;
      T     LW 8;
      CDB;
      OPN   DI [LW 8];
      TAR2  LD 4;
      +AR2  P#1784.0;
      UC    FB 19;
      LAR2  LD 4;
      CDB;
      BLD   15;
NETWORK
TITLE = =A-3126-TSC01_AP : ACT. POWER FAN 2 FU 
      NOP   0;
//-InLocal---
      A     #tmpLocal;
      O     DB922.DBX 1569.1;	// emergency regime without fan 2
      =     DIX [AR2,P#1875.4];
//-Monitoring--- 
      CLR;
      =     DIX [AR2,P#1874.0];
      CLR;
      =     DIX [AR2,P#1874.1];
      CLR;
      =     DIX [AR2,P#1874.2];
      CLR;
      =     DIX [AR2,P#1874.3];
      CLR;
      =     DIX [AR2,P#1874.4];
// 
//-Read inputs---
//MW 2010.04.09      L     #A_3126_TSC01_COM.Output.SetpointValue01
//MW 2010.04.09      ITD   
//MW 2010.04.09      DTR   
//MW 2010.04.09      ABS   
//MW 2010.04.09      RND   
      L     DIW [AR2,P#1670.0];
      T     DIW [AR2,P#1878.0];
      A     DB50.DBX 32.3;
      =     DIX [AR2,P#1875.0];
// 
//-Set Parameters---
// 
//-Call object control---
      BLD   14;
// 
//-Write outputs---
      =     L 10.0;
      L     DINO;
      T     LW 8;
      CDB;
      OPN   DI [LW 8];
      TAR2  LD 4;
      +AR2  P#1872.0;
      UC    FB 19;
      LAR2  LD 4;
      CDB;
      BLD   15;
NETWORK
TITLE = =A-3126-TSC01_AT : ACT. TORQUE FAN 2 FU 
      NOP   0;
//-InLocal---
      A     #tmpLocal;
      O     DB922.DBX 1569.1;	// emergency regime without fan 2
      =     DIX [AR2,P#1963.4];
//-Monitoring--- 
      CLR;
      =     DIX [AR2,P#1962.0];
      CLR;
      =     DIX [AR2,P#1962.1];
      CLR;
      =     DIX [AR2,P#1962.2];
      CLR;
      =     DIX [AR2,P#1962.3];
      CLR;
      =     DIX [AR2,P#1962.4];
// 
//-Read inputs---
//MW 2010.04.09      L     #A_3126_TSC01_COM.Output.SetpointValue01
//MW 2010.04.09      ITD   
//MW 2010.04.09      DTR   
//MW 2010.04.09      ABS   
//MW 2010.04.09      RND   
      L     DIW [AR2,P#1668.0];
      T     DIW [AR2,P#1966.0];
      A     DB50.DBX 32.3;
      =     DIX [AR2,P#1963.0];
// 
//-Set Parameters---
// 
//-Call object control---
      BLD   14;
// 
//-Write outputs---
      =     L 10.0;
      L     DINO;
      T     LW 8;
      CDB;
      OPN   DI [LW 8];
      TAR2  LD 4;
      +AR2  P#1960.0;
      UC    FB 19;
      LAR2  LD 4;
      CDB;
      BLD   15;
NETWORK
TITLE = =A-3125-TSC01 : FAN 1 FU KOMMUNIKATION
      NOP   0;
//-InLocal---
      A     #tmpLocal;
      =     DIX [AR2,P#2051.4];
// 
//-Monitoring---
      CLR;
      =     DIX [AR2,P#2050.0];
      CLR;
      =     DIX [AR2,P#2050.1];
// 
//-PreAlarm---
      CLR;
      =     DIX [AR2,P#2050.2];
      CLR;
      =     DIX [AR2,P#2050.3];
// 
//-Additional commands---
//      CLR
//      S     #A_3125_TSC01.CmdRunTimeOutTime
// 
//-Read inputs---
//MW 2010.04.09    U     "ENG_RemarkFlag"
      A     DIX [AR2,P#668.1];
      A     DIX [AR2,P#669.1];
      AN    DIX [AR2,P#669.3];
      =     DIX [AR2,P#2050.6];
// 
//-Set Parameters---
// 
//-Call object control---
      BLD   14;
// 
//-Write outputs---
      =     L 10.0;
      L     DINO;
      T     LW 8;
      CDB;
      OPN   DI [LW 8];
      TAR2  LD 4;
      +AR2  P#2048.0;
      UC    FB 14;
      LAR2  LD 4;
      CDB;
      BLD   15;
NETWORK
TITLE = =A-3126-TSC01 : FAN 2 FU KOMMUNIKATION
      NOP   0;
//-InLocal---
      A     #tmpLocal;
      =     DIX [AR2,P#2085.4];
// 
//-Monitoring---
      CLR;
      =     DIX [AR2,P#2084.0];
      CLR;
      =     DIX [AR2,P#2084.1];
// 
//-PreAlarm---
      CLR;
      =     DIX [AR2,P#2084.2];
      CLR;
      =     DIX [AR2,P#2084.3];
// 
//-Additional commands---
//      CLR
//      S     #A_3126_TSC01.CmdRunTimeOutTime
// 
//-Read inputs---
//MW 2010.04.09    U     "ENG_RemarkFlag"
      A     DIX [AR2,P#1662.1];
      A     DIX [AR2,P#1663.1];
      AN    DIX [AR2,P#1663.3];
      =     DIX [AR2,P#2084.6];
// 
//-Set Parameters---
// 
//-Call object control---
      BLD   14;
// 
//-Write outputs---
      =     L 10.0;
      L     DINO;
      T     LW 8;
      CDB;
      OPN   DI [LW 8];
      TAR2  LD 4;
      +AR2  P#2082.0;
      UC    FB 14;
      LAR2  LD 4;
      CDB;
      BLD   15;
NETWORK
TITLE = Test Fault
      A     DIX [AR2,P#65.7];
      O     DIX [AR2,P#153.7];
      O     DIX [AR2,P#241.7];
      O     DIX [AR2,P#329.7];
      O     DIX [AR2,P#417.4];
      O     DIX [AR2,P#707.7];
      O     DIX [AR2,P#795.7];
      O     DIX [AR2,P#883.7];
      O     DIX [AR2,P#971.7];
      O     DIX [AR2,P#1059.7];
      O     DIX [AR2,P#1147.7];
      O     DIX [AR2,P#1235.7];
      O     DIX [AR2,P#1323.7];
      O     DIX [AR2,P#1411.4];
      O     DIX [AR2,P#1701.7];
      O     DIX [AR2,P#1789.7];
      O     DIX [AR2,P#1877.7];
      O     DIX [AR2,P#1965.7];
      O     DIX [AR2,P#2053.4];
      O     DIX [AR2,P#2087.4];
      =     DIX [AR2,P#19.2];
NETWORK
TITLE = Test Warning
      A     DIX [AR2,P#65.6];
      O     DIX [AR2,P#153.6];
      O     DIX [AR2,P#241.6];
      O     DIX [AR2,P#329.6];
      O     DIX [AR2,P#707.6];
      O     DIX [AR2,P#795.6];
      O     DIX [AR2,P#883.6];
      O     DIX [AR2,P#971.6];
      O     DIX [AR2,P#1059.6];
      O     DIX [AR2,P#1147.6];
      O     DIX [AR2,P#1235.6];
      O     DIX [AR2,P#1323.6];
      O     DIX [AR2,P#1701.6];
      O     DIX [AR2,P#1789.6];
      O     DIX [AR2,P#1877.6];
      O     DIX [AR2,P#1965.6];
      =     DIX [AR2,P#17.6];
NETWORK
TITLE = Test Stopped
      A     DIX [AR2,P#417.0];
      A     DIX [AR2,P#1411.0];
      AN    DIX [AR2,P#19.2];
      =     DIX [AR2,P#19.0];
NETWORK
TITLE = Test Started
      A(;
      A     DIX [AR2,P#417.2];
      O     DB922.DBX 1569.0;	// emergency regime without fan 1
      );
      A(;
      A     DIX [AR2,P#1411.2];
      O     DB922.DBX 1569.1;	// emergency regime without fan 2
      );
      AN    DIX [AR2,P#19.0];
      AN    DIX [AR2,P#19.2];
      =     DIX [AR2,P#19.1];
NETWORK
TITLE = Enable Previous Group
//MW 2010.04.09    U     #Gr.VarStarted
      A     DIX [AR2,P#417.2];
      A     DIX [AR2,P#794.1];	// InpValue>=ParL
      A     DIX [AR2,P#1411.2];
      A     DIX [AR2,P#1788.1];	// InpValue>=ParL
      O;
      A     DIX [AR2,P#417.2];
      A     DIX [AR2,P#794.2];	// InpValue>=ParH
      O;
      A     DIX [AR2,P#1411.2];
      A     DIX [AR2,P#1788.2];	// InpValue>=ParH
      =     DIX [AR2,P#18.7];
NETWORK
TITLE = Call Methode State
//1. Make State of the group: This function use the signals:
//        Gr.VarStopped, Gr.VarStarted, Gr.VarFault
//2.Reset Commands to group: e.g.CmdFaultReset
      BLD   14;
      =     L 10.0;
      L     DINO;
      T     LW 8;
      CDB;
      OPN   DI [LW 8];
      TAR2  LD 4;
      L     2;
      T     DIW [AR2,P#0.0];
      +AR2  P#0.0;
      UC    FB 10;
      LAR2  LD 4;
      CDB;
      BLD   15;
NETWORK
TITLE = Init
      SET;
      R     DIX [AR2,P#58.2];
      R     DIX [AR2,P#58.3];
NETWORK
TITLE = Write data to group control
      A     DIX [AR2,P#17.0];
      =     DB9.DBX 483.6;
      A     DIX [AR2,P#17.2];
      =     DB9.DBX 523.6;
      A     DIX [AR2,P#17.4];
      =     DB9.DBX 563.6;
      A     DIX [AR2,P#17.6];
      =     DB9.DBX 603.6;
      A     DIX [AR2,P#18.5];
      =     DB9.DBX 643.6;
      A     DIX [AR2,P#18.2];
      =     DB9.DBX 883.6;
      A     DIX [AR2,P#18.3];
      =     DB9.DBX 843.6;
      A     DIX [AR2,P#17.5];
      =     DB9.DBX 803.6;
      A     DIX [AR2,P#18.4];
      =     DB9.DBX 923.6;
      A     DIX [AR2,P#19.3];
      =     DB9.DBX 963.6;
NETWORK
TITLE = End of block
      BE;
END_FUNCTION_BLOCK

